PROGRAM StationVisualProgram
VAR
	
	
	(* These are all used for animating the different positions of the cylinder bases *)
	MagPos1: BOOL := TRUE;
	MagPos2: BOOL := TRUE;
	MagPos3: BOOL := TRUE;
	MagPos4: BOOL := TRUE;
	MagPos5: BOOL := TRUE;
	BasePos6: BOOL := TRUE;
	BasePos7: BOOL :=  TRUE;
	BasePos7a: BOOL := TRUE;
	BasePos7b: BOOL := TRUE;
	BasePos7c: BOOL := TRUE;
	BasePos7d: BOOL := TRUE;
	BasePos7e: BOOL := TRUE;
	BasePos8: BOOL := TRUE;
	BasePos8a: BOOL := TRUE;
	BasePos8b: BOOL := TRUE;
	
	(*Used to animate the pusher of the testing station*)
	EjecCylDown: BOOL := TRUE;
	EjecCylUp: BOOL := TRUE;
	
	(* These timers are used to imitate the moving time in the visualization*)
	T_hMeas: TIME := TIME#1S500MS;
	t_half: TIME := TIME#250MS;
	TON_0: TON;
	TON_1: TON;
	TON_2: TON;
	TON_3: TON;
	TON_4: TON;
	TON_5: TON;
	TON_6: TON;
	TON_7: TON;
	TON_8: TON;
	TON_9: TON;
	
	(* These are just used to maintain the sequence or flow*)
	keep1: BOOL;
	next2: BOOL;
	Next3: BOOL;	
	Dummy: BOOL;
	
	H_MeasCylDo: BOOL := TRUE; (*Used to animate the measuring actuator*)
	
END_VAR
VAR // added by the converter: edge detectors and wires of the graphical bodies
    _w1, _w2, _w3, _w4, _w5, _w6, _w7, _w8, _w9, _w10, _w11, _w12, _w13, _w14, _w15, _w16, _w17, _w18, _w19, _w20 : BOOL;
END_VAR

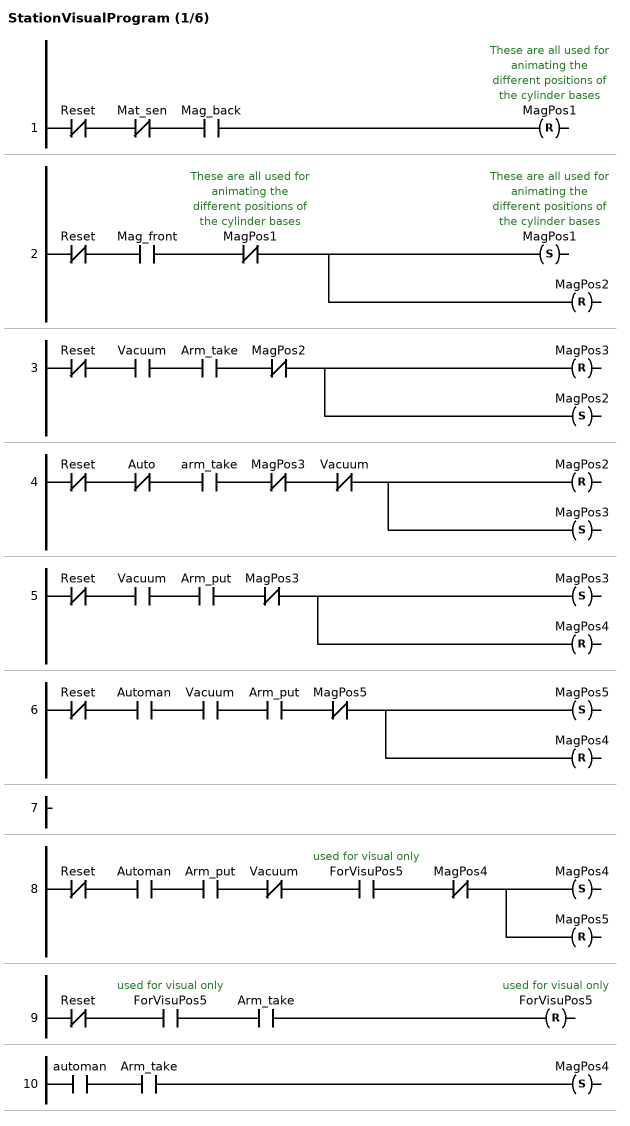
// NETWORK 1
//   MagPos1: These are all used for animating the different positions of the cylinder bases
MagPos1 R= NOT Reset AND NOT Mat_sen AND Mag_back;

// NETWORK 2
//   MagPos1: These are all used for animating the different positions of the cylinder bases
_w1 := NOT Reset AND Mag_front AND NOT MagPos1;
MagPos1 S= _w1;
MagPos2 R= _w1;

// NETWORK 3
_w2 := NOT Reset AND Vacuum AND Arm_take AND NOT MagPos2;
MagPos3 R= _w2;
MagPos2 S= _w2;

// NETWORK 4
_w3 := NOT Reset AND NOT Auto AND arm_take AND NOT MagPos3 AND NOT Vacuum;
MagPos2 R= _w3;
MagPos3 S= _w3;

// NETWORK 5
_w4 := NOT Reset AND Vacuum AND Arm_put AND NOT MagPos3;
MagPos3 S= _w4;
MagPos4 R= _w4;

// NETWORK 6
_w5 := NOT Reset AND Automan AND Vacuum AND Arm_put AND NOT MagPos5;
MagPos5 S= _w5;
MagPos4 R= _w5;

// NETWORK 7

// NETWORK 8
//   ForVisuPos5: used for visual only
_w6 := NOT Reset AND Automan AND Arm_put AND NOT Vacuum AND ForVisuPos5 AND NOT MagPos4;
MagPos4 S= _w6;
MagPos5 R= _w6;

// NETWORK 9
//   ForVisuPos5: used for visual only
ForVisuPos5 R= NOT Reset AND ForVisuPos5 AND Arm_take;

// NETWORK 10
MagPos4 S= automan AND Arm_take;

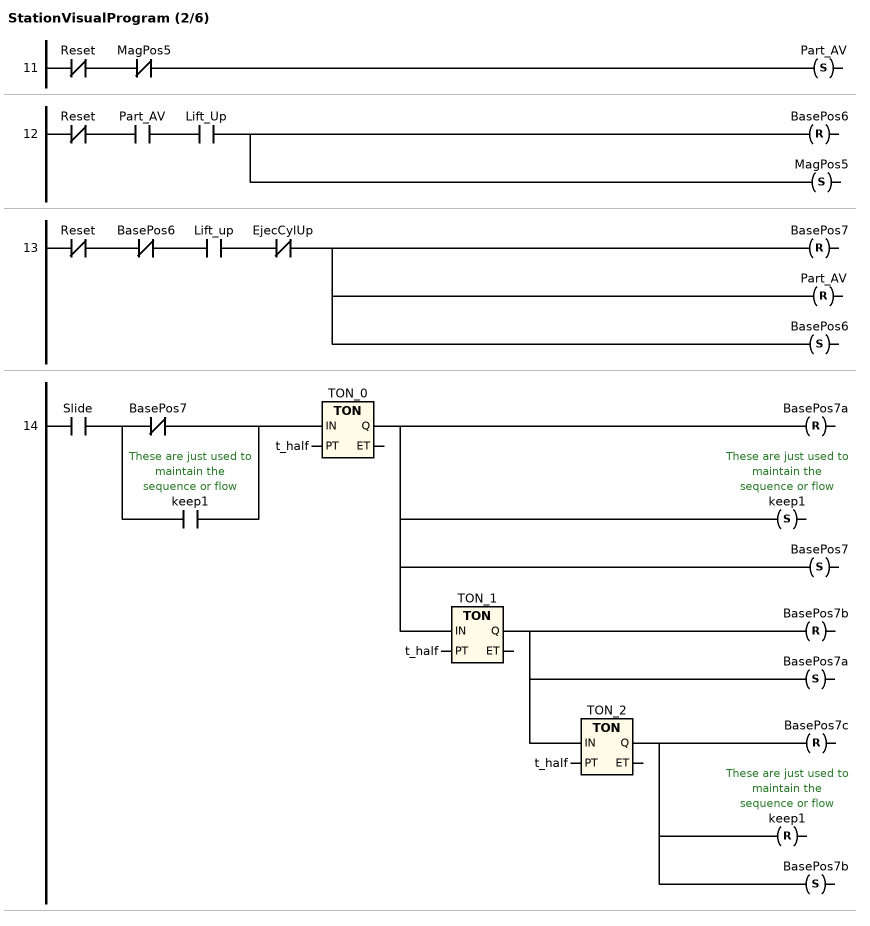
// NETWORK 11
Part_AV S= NOT Reset AND NOT MagPos5;

// NETWORK 12
_w7 := NOT Reset AND Part_AV AND Lift_Up;
BasePos6 R= _w7;
MagPos5 S= _w7;

// NETWORK 13
_w8 := NOT Reset AND NOT BasePos6 AND Lift_up AND NOT EjecCylUp;
BasePos7 R= _w8;
Part_AV R= _w8;
BasePos6 S= _w8;

// NETWORK 14
//   keep1: These are just used to maintain the sequence or flow
TON_0(IN := Slide AND (NOT BasePos7 OR keep1), PT := t_half); // TON
BasePos7a R= TON_0.Q;
keep1 S= TON_0.Q;
BasePos7 S= TON_0.Q;
TON_1(IN := TON_0.Q, PT := t_half); // TON
BasePos7b R= TON_1.Q;
BasePos7a S= TON_1.Q;
TON_2(IN := TON_1.Q, PT := t_half); // TON
BasePos7c R= TON_2.Q;
keep1 R= TON_2.Q;
BasePos7b S= TON_2.Q;

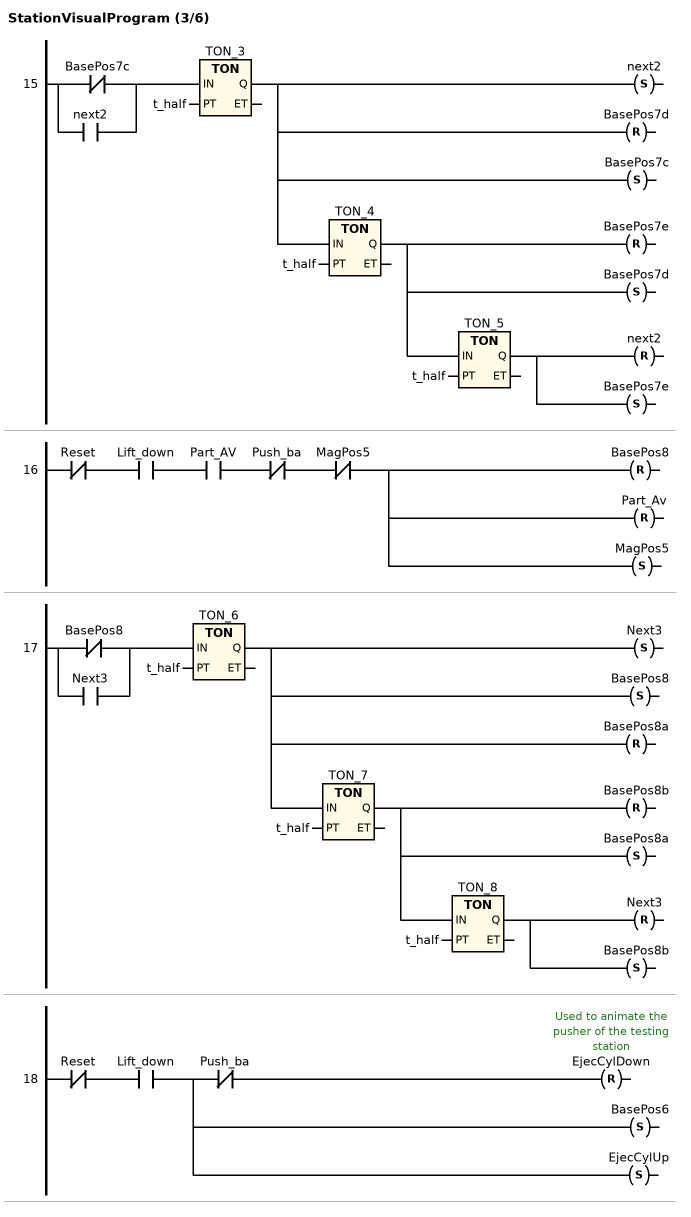
// NETWORK 15
TON_3(IN := NOT BasePos7c OR next2, PT := t_half); // TON
next2 S= TON_3.Q;
BasePos7d R= TON_3.Q;
BasePos7c S= TON_3.Q;
TON_4(IN := TON_3.Q, PT := t_half); // TON
BasePos7e R= TON_4.Q;
BasePos7d S= TON_4.Q;
TON_5(IN := TON_4.Q, PT := t_half); // TON
next2 R= TON_5.Q;
BasePos7e S= TON_5.Q;

// NETWORK 16
_w9 := NOT Reset AND Lift_down AND Part_AV AND NOT Push_ba AND NOT MagPos5;
BasePos8 R= _w9;
Part_Av R= _w9;
MagPos5 S= _w9;

// NETWORK 17
TON_6(IN := NOT BasePos8 OR Next3, PT := t_half); // TON
Next3 S= TON_6.Q;
BasePos8 S= TON_6.Q;
BasePos8a R= TON_6.Q;
TON_7(IN := TON_6.Q, PT := t_half); // TON
BasePos8b R= TON_7.Q;
BasePos8a S= TON_7.Q;
TON_8(IN := TON_7.Q, PT := t_half); // TON
Next3 R= TON_8.Q;
BasePos8b S= TON_8.Q;

// NETWORK 18
//   EjecCylDown: Used to animate the pusher of the testing station
_w10 := NOT Reset AND Lift_down;
EjecCylDown R= _w10 AND NOT Push_ba;
BasePos6 S= _w10;
EjecCylUp S= _w10;

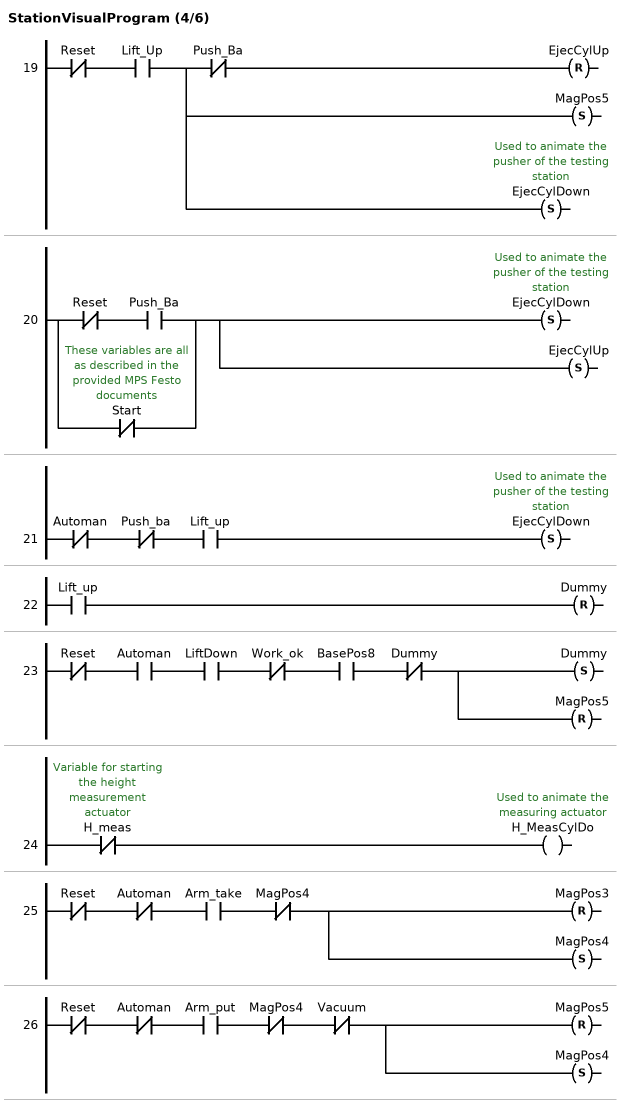
// NETWORK 19
//   EjecCylDown: Used to animate the pusher of the testing station
_w11 := NOT Reset AND Lift_Up;
EjecCylUp R= _w11 AND NOT Push_Ba;
MagPos5 S= _w11;
EjecCylDown S= _w11;

// NETWORK 20
//   Start: These variables are all as described in the provided MPS Festo documents
//   EjecCylDown: Used to animate the pusher of the testing station
_w12 := NOT Reset AND Push_Ba OR NOT Start;
EjecCylDown S= _w12;
EjecCylUp S= _w12;

// NETWORK 21
//   EjecCylDown: Used to animate the pusher of the testing station
EjecCylDown S= NOT Automan AND NOT Push_ba AND Lift_up;

// NETWORK 22
Dummy R= Lift_up;

// NETWORK 23
_w13 := NOT Reset AND Automan AND LiftDown AND NOT Work_ok AND BasePos8 AND NOT Dummy;
Dummy S= _w13;
MagPos5 R= _w13;

// NETWORK 24
//   H_meas: Variable for starting the height measurement actuator
//   H_MeasCylDo: Used to animate the measuring actuator
H_MeasCylDo := NOT H_meas;

// NETWORK 25
_w14 := NOT Reset AND NOT Automan AND Arm_take AND NOT MagPos4;
MagPos3 R= _w14;
MagPos4 S= _w14;

// NETWORK 26
_w15 := NOT Reset AND NOT Automan AND Arm_put AND NOT MagPos4 AND NOT Vacuum;
MagPos5 R= _w15;
MagPos4 S= _w15;

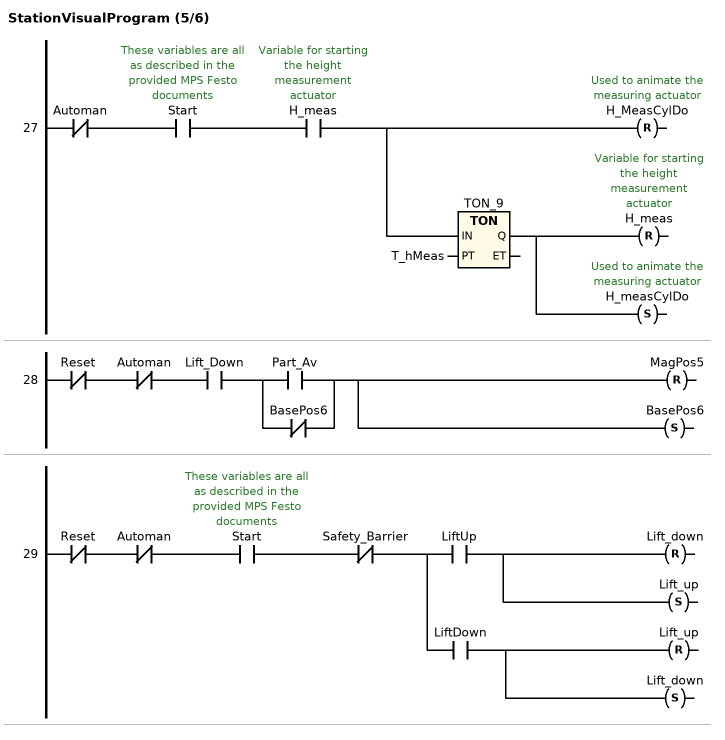
// NETWORK 27
//   Start: These variables are all as described in the provided MPS Festo documents
//   H_meas: Variable for starting the height measurement actuator
//   H_MeasCylDo: Used to animate the measuring actuator
//   T_hMeas: These timers are used to imitate the moving time in the visualization
//   H_measCylDo: Used to animate the measuring actuator
_w16 := NOT Automan AND Start AND H_meas;
H_MeasCylDo R= _w16;
TON_9(IN := _w16, PT := T_hMeas); // TON
H_meas R= TON_9.Q;
H_measCylDo S= TON_9.Q;

// NETWORK 28
_w17 := NOT Reset AND NOT Automan AND Lift_Down AND (Part_Av OR NOT BasePos6);
MagPos5 R= _w17;
BasePos6 S= _w17;

// NETWORK 29
//   Start: These variables are all as described in the provided MPS Festo documents
_w18 := NOT Reset AND NOT Automan AND Start AND NOT Safety_Barrier;
_w19 := _w18 AND LiftUp;
Lift_down R= _w19;
Lift_up S= _w19;
_w20 := _w18 AND LiftDown;
Lift_up R= _w20;
Lift_down S= _w20;

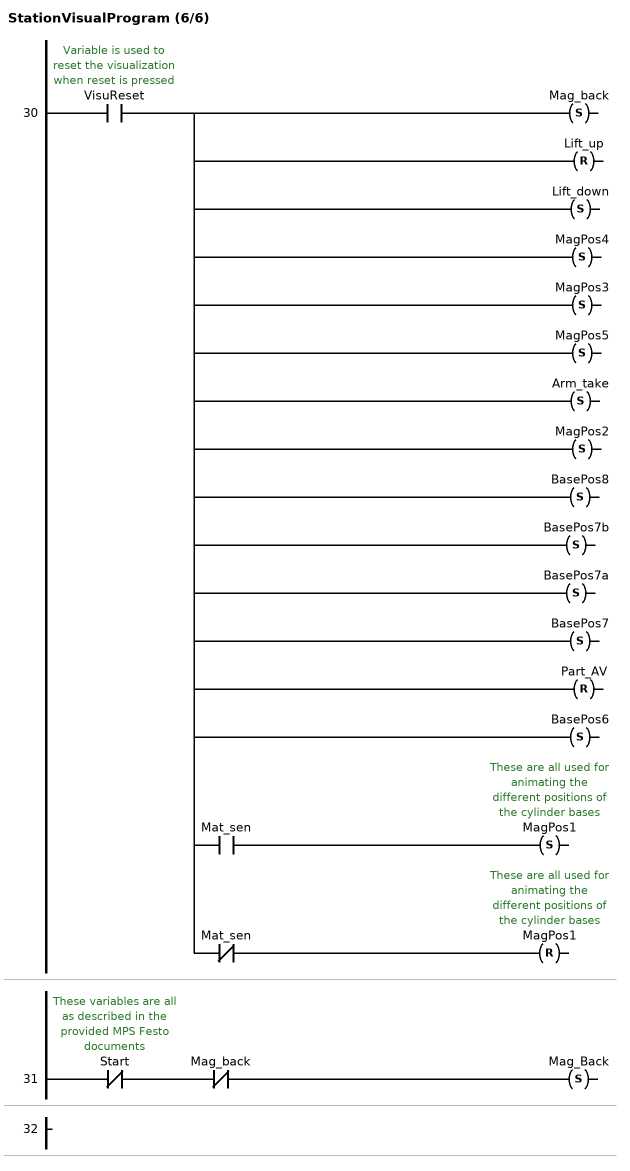
// NETWORK 30
//   VisuReset: Variable is used to reset the visualization when reset is pressed
//   MagPos1: These are all used for animating the different positions of the cylinder bases
Mag_back S= VisuReset;
Lift_up R= VisuReset;
Lift_down S= VisuReset;
MagPos4 S= VisuReset;
MagPos3 S= VisuReset;
MagPos5 S= VisuReset;
Arm_take S= VisuReset;
MagPos2 S= VisuReset;
BasePos8 S= VisuReset;
BasePos7b S= VisuReset;
BasePos7a S= VisuReset;
BasePos7 S= VisuReset;
Part_AV R= VisuReset;
BasePos6 S= VisuReset;
MagPos1 S= VisuReset AND Mat_sen;
MagPos1 R= VisuReset AND NOT Mat_sen;

// NETWORK 31
//   Start: These variables are all as described in the provided MPS Festo documents
Mag_Back S= NOT Start AND NOT Mag_back;

// NETWORK 32

END_PROGRAM

(* stored: Version 1.1.0.1, ProductVersion 3.1.4018.5
   POU StationVisualProgram: Id {7f81ac29-a387-495f-8c45-8b8bed2fcdd2}, SpecialFunc None *)
